{attribute 'qualified_only'}
VAR_GLOBAL
END_VAR

(* stored: Version 1.1.0.1, ProductVersion 3.1.4024.12
   GVL GVL_SUBSTATION: Id {b6a00a5c-1184-4cfa-a782-9273f872f113} *)
